// TIA Portal project "SCL EJERCICIO 1" (V11)

(* hardware
DEVICE "S7300/ET200 station_1"  SIMATIC 300-Station
   slot 0: "Perfil soporte_0"  Rail  6ES7 390-1***0-0AA0
   slot 2: "PLC_1"  CPU 313C-2 DP  6ES7 313-6CF03-0AB0  V2.6
      slot 0: "Interfaz MPI_1"  MPI
      slot 1: "Interfaz DP_1"  DP
      slot 2: "DI16/DO16_1"  DI16/DO16
      slot 4: "Contaje_1"  Counter
*)

// ===== PLC "PLC_1"  CPU 313C-2 DP =====

VAR_GLOBAL   // PLC tag table "Tabla de variables estándar"
   "Tag_1" AT %E0.0 : Bool;
   "Tag_2" AT %E0.1 : Bool;
   "Tag_3" AT %E0.2 : Bool;
   "Tag_4" AT %E0.3 : Bool;
   "Tag_5" AT %A0.0 : Bool;
   "Tag_6" AT %A0.1 : Bool;
   "Tag_7" AT %A0.2 : Bool;
   "Tag_8" AT %A0.3 : Bool;
   "Tag_9" AT %A0.4 : Bool;
   "Tag_10" AT %A0.5 : Bool;
END_VAR

DATA_BLOCK "INVERSION DE GIRO_DB"   // DB1
{ S7_Optimized_Access := 'FALSE' }
VERSION : 0.1
// stored: InstanceOfName INVERSION DE GIRO
"INVERSION DE GIRO"
BEGIN
END_DATA_BLOCK

FUNCTION_BLOCK "INVERSION DE GIRO"   // FB1, SCL
{ S7_Optimized_Access := 'FALSE' }
VERSION : 0.1
   VAR_INPUT
      PARO : Bool;
      DERERCHA : Bool;
      IZQUIERDA : Bool;
      "RELE TERMICO" : Bool;
   END_VAR
   VAR_OUTPUT
      "MARCHA DERECHA" : Bool;
      "LED DERECHA" : Bool;
      "MARCHA IZQUIERDA" : Bool;
      "LED IZQUIERDA" : Bool;
      "LED PARO" : Bool;
      "LED AVERIA" : Bool;
   END_VAR
BEGIN
   IF #PARO THEN (* condiciones de paro cuado este activo no funciona nada esceoto led paro * *)
     #"LED PARO" := TRUE ;
     #"MARCHA DERECHA":=FALSE;
     #"LED DERECHA":=FALSE;
     #"MARCHA IZQUIERDA":=FALSE;
     #"LED IZQUIERDA":=FALSE;
      END_IF;

   IF NOT  #"MARCHA DERECHA" AND NOT #"MARCHA IZQUIERDA" THEN (* led #PARO *)
     #"LED PARO":=TRUE;
      END_IF;

   IF #DERERCHA AND   #"LED PARO" AND NOT #PARO AND NOT #"RELE TERMICO" AND NOT #"MARCHA IZQUIERDA" THEN (* condiciones marcha derecha y led derecha *)
     #"MARCHA DERECHA":= TRUE;
     #"MARCHA IZQUIERDA":=FALSE ;
     #"LED DERECHA":=TRUE ;
     #"LED IZQUIERDA":=FALSE;
     #"LED PARO":= FALSE;
     #"LED AVERIA":=false;
     END_IF;

   IF #IZQUIERDA AND   #"LED PARO"  AND NOT #PARO AND NOT #"RELE TERMICO" AND NOT #"MARCHA IZQUIERDA" THEN (* condiciones marcha izquierda y led izquierda *)
     #"MARCHA IZQUIERDA":=TRUE;
     #"LED IZQUIERDA":=TRUE ;
     #"MARCHA DERECHA":=FALSE;
     #"LED DERECHA" := FALSE ;
     #"LED PARO":=false ;
     #"LED AVERIA":=false;
   END_IF;

   IF #"RELE TERMICO" THEN (* disparo termico mientras que este activo no funciona nada salvo led paro y averia *)
     #"MARCHA DERECHA":=false;
     #"LED DERECHA":=false;
     #"MARCHA IZQUIERDA":=false;
     #"LED IZQUIERDA":=false;
     #"LED AVERIA":=true;
     #"LED PARO":=true;
   ELSE
     #"LED AVERIA":=false;
   END_IF;
END_FUNCTION_BLOCK

ORGANIZATION_BLOCK "Main"   // OB1, LAD
TITLE = "Main Program Sweep (Cycle)"
{ S7_Optimized_Access := 'FALSE' }
VERSION : 0.1
   VAR_TEMP
      OB1_EV_CLASS : Byte;   // Bits 0-3 = 1 (Coming event), Bits 4-7 = 1 (Event class 1)
      OB1_SCAN_1 : Byte;   // 1 (Cold restart scan 1 of OB 1), 3 (Scan 2-n of OB 1)
      OB1_PRIORITY : Byte;   // Priority of OB Execution
      OB1_OB_NUMBR : Byte;   // 1 (Organization block 1, OB1)
      OB1_RESERVED_1 : Byte;   // Reserved for system
      OB1_RESERVED_2 : Byte;   // Reserved for system
      OB1_PREV_CYCLE : Int;   // Cycle time of previous OB1 scan (milliseconds)
      OB1_MIN_CYCLE : Int;   // Minimum cycle time of OB1 (milliseconds)
      OB1_MAX_CYCLE : Int;   // Maximum cycle time of OB1 (milliseconds)
      OB1_DATE_TIME : Date_And_Time;   // Date and time OB1 started
   END_VAR
BEGIN

REGION Network 1
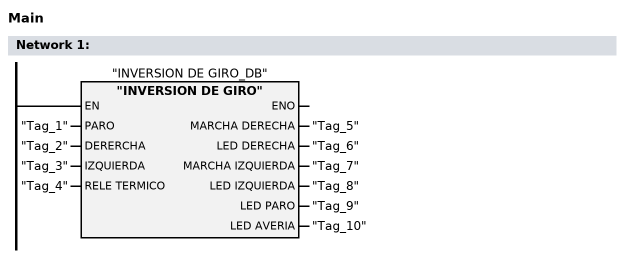
   RUNG wire#powerrail
      "INVERSION DE GIRO_DB"(PARO := "Tag_1", DERERCHA := "Tag_2", IZQUIERDA := "Tag_3", "RELE TERMICO" := "Tag_4", "MARCHA DERECHA" => "Tag_5", "LED DERECHA" => "Tag_6", "MARCHA IZQUIERDA" => "Tag_7", "LED IZQUIERDA" => "Tag_8", "LED PARO" => "Tag_9", "LED AVERIA" => "Tag_10")
   END_RUNG
   // the same network as SCL:
   "INVERSION DE GIRO_DB"(PARO := "Tag_1",   // "INVERSION DE GIRO"
                          DERERCHA := "Tag_2",
                          IZQUIERDA := "Tag_3",
                          "RELE TERMICO" := "Tag_4",
                          "MARCHA DERECHA" => "Tag_5",
                          "LED DERECHA" => "Tag_6",
                          "MARCHA IZQUIERDA" => "Tag_7",
                          "LED IZQUIERDA" => "Tag_8",
                          "LED PARO" => "Tag_9",
                          "LED AVERIA" => "Tag_10");
END_REGION
END_ORGANIZATION_BLOCK